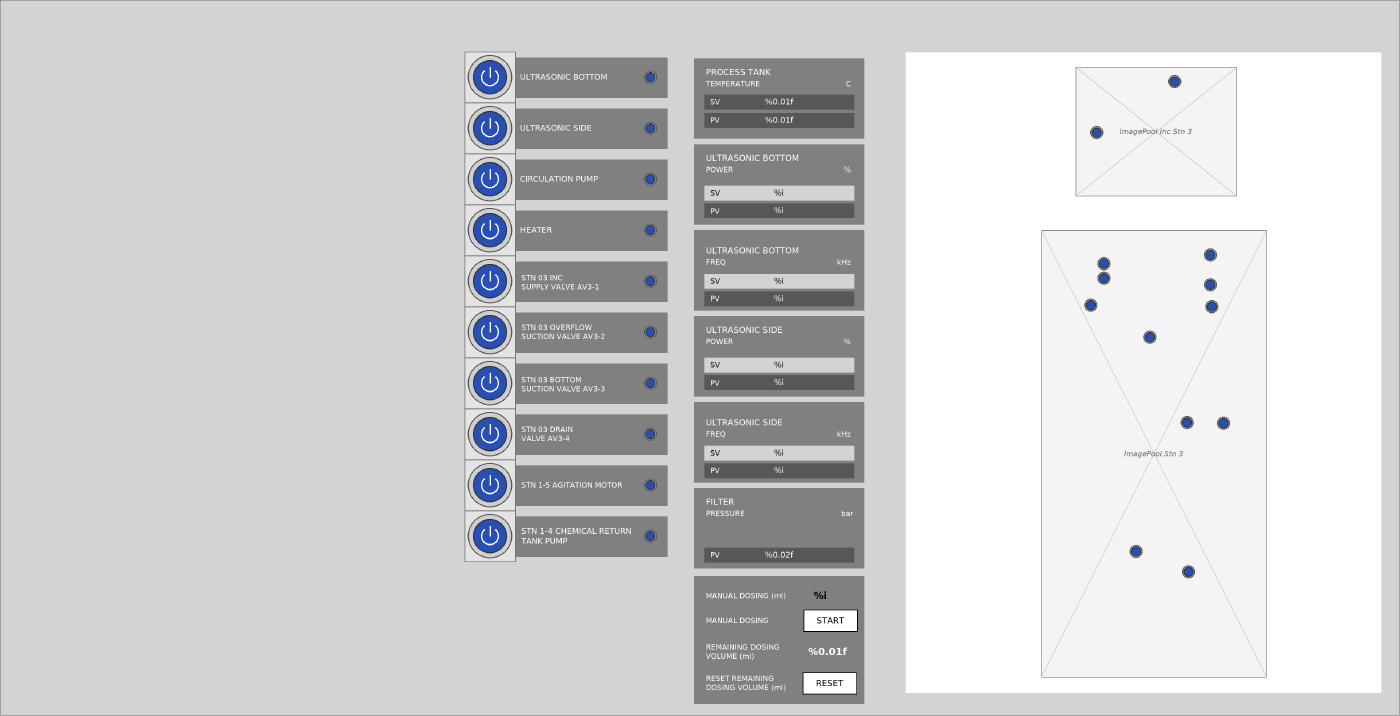
VISUALIZATION Manual_Station03  // 1920x983
    Rectangle (0,0 1920x983)
    Rectangle (1242,72 652x879)
    Image (1428,316 309x614), image: ImagePool.Stn 3
    RoundedRectangle (676,79 239x55)
    Label (710,98 163x16), "ULTRASONIC BOTTOM"
    Lamp1 (882,96 20x20), variable: ARdsMAP_HmiVariableStn[3].bProTankUsBtm_IND, style: Lamp-Lamp1-Blue
    PowerSwitch (637,71 70x70), variable: ARdsMAP_HmiVariableStn[3].bProTankUsBtm_PB, behaviour: TOGGLE, style: Switch-PowerSwitch-Blue
    RoundedRectangle (684,219 231x55)
    Label (710,238 151x16), "CIRCULATION PUMP"
    Lamp1 (882,236 20x20), variable: ARdsMAP_HmiVariableStn[3].bProTankPump_IND, style: Lamp-Lamp1-Blue
    PowerSwitch (637,211 70x70), variable: ARdsMAP_HmiVariableStn[3].bProTankPump_PB, behaviour: TOGGLE, style: Switch-PowerSwitch-Blue
    RoundedRectangle (684,289 231x55)
    Label (710,308 151x16), "HEATER"
    Lamp1 (882,306 20x20), variable: ARdsMAP_HmiVariableStn[3].bProTankHeater_IND, style: Lamp-Lamp1-Blue
    PowerSwitch (637,281 70x70), variable: ARdsMAP_HmiVariableStn[3].bProTankHeater_PB, behaviour: TOGGLE, style: Switch-PowerSwitch-Blue
    RoundedRectangle (676,149 239x55)
    Label (710,168 163x16), "ULTRASONIC SIDE"
    Lamp1 (882,166 20x20), variable: ARdsMAP_HmiVariableStn[3].bProTankUsSide_IND, style: Lamp-Lamp1-Blue
    PowerSwitch (637,141 70x70), variable: ARdsMAP_HmiVariableStn[3].bProTankUsSide_PB, behaviour: TOGGLE, style: Switch-PowerSwitch-Blue
    RoundedRectangle (684,429 231x55)
    Label (712,438 160x36), "STN 03 OVERFLOW SUCTION VALVE AV3-2"
    Lamp1 (882,446 20x20), variable: ARdsMAP_HmiVariableStn[3].bValve02_IND, style: Lamp-Lamp1-Blue
    PowerSwitch (637,421 70x70), variable: ARdsMAP_HmiVariableStn[3].bValve02_PB, behaviour: TOGGLE, style: Switch-PowerSwitch-Blue
    RoundedRectangle (684,359 231x55)
    Lamp1 (882,376 20x20), variable: ARdsMAP_HmiVariableStn[3].bValve01_IND, style: Lamp-Lamp1-Blue
    PowerSwitch (637,351 70x70), variable: ARdsMAP_HmiVariableStn[3].bValve01_PB, behaviour: TOGGLE, style: Switch-PowerSwitch-Blue
    Label (712,370 151x36), "STN 03 INC SUPPLY VALVE AV3-1"
    RoundedRectangle (684,569 231x55)
    Label (712,578 160x36), "STN 03 DRAIN VALVE AV3-4"
    Lamp1 (882,586 20x20), variable: ARdsMAP_HmiVariableStn[3].bValve04_IND, style: Lamp-Lamp1-Blue
    PowerSwitch (637,561 70x70), variable: ARdsMAP_HmiVariableStn[3].bValve04_PB, behaviour: TOGGLE, style: Switch-PowerSwitch-Blue
    RoundedRectangle (684,499 231x55)
    Lamp1 (882,516 20x20), variable: ARdsMAP_HmiVariableStn[3].bValve03_IND, style: Lamp-Lamp1-Blue
    PowerSwitch (637,491 70x70), variable: ARdsMAP_HmiVariableStn[3].bValve03_PB, behaviour: TOGGLE, style: Switch-PowerSwitch-Blue
    Label (712,510 151x36), "STN 03 BOTTOM SUCTION VALVE AV3-3"
    RoundedRectangle (684,639 231x55)
    Label (712,648 160x36), "STN 1-5 AGITATION MOTOR"
    Lamp1 (882,656 20x20), variable: ARdsMAP_HmiVariableGeneral.bProTankAgitationMotor_IND, style: Lamp-Lamp1-Blue
    PowerSwitch (637,631 70x70), variable: ARdsMAP_HmiVariableGeneral.bProTankAgitationMotor_PB, behaviour: TOGGLE, style: Switch-PowerSwitch-Blue
    RoundedRectangle (684,709 231x55)
    Label (712,718 160x36), "STN 1-4 CHEMICAL RETURN TANK PUMP"
    Lamp1 (882,726 20x20), variable: ARdsMAP_HmiVariableGeneral.bProTankPump_IND, style: Lamp-Lamp1-Blue
    PowerSwitch (637,701 70x70), variable: ARdsMAP_HmiVariableGeneral.bProTankPump_PB, behaviour: TOGGLE, style: Switch-PowerSwitch-Blue
    Lamp1 (1567,453 20x20), variable: ARdsMAP_HmiVariableStn[3].bProTankUsBtm_IND, style: Lamp-Lamp1-Blue
    Lamp1 (1548,747 20x20), variable: ARdsMAP_HmiVariableStn[3].bProTankPump_IND, style: Lamp-Lamp1-Blue
    Lamp1 (1504,372 20x20), variable: ARdsMAP_HmiVariableStn[3].bProTankHeater_IND, style: Lamp-Lamp1-Blue
    Lamp1 (1486,409 20x20), variable: ARdsMAP_HmiVariableStn[3].bProTankUsSide_IND, style: Lamp-Lamp1-Blue
    Lamp1 (1668,571 20x20), variable: ARdsMAP_HmiVariableStn[3].bValve02_IND, style: Lamp-Lamp1-Blue
    Lamp1 (1620,775 20x20), variable: ARdsMAP_HmiVariableStn[3].bValve04_IND, style: Lamp-Lamp1-Blue
    Lamp1 (1618,570 20x20), variable: ARdsMAP_HmiVariableStn[3].bValve03_IND, style: Lamp-Lamp1-Blue
    Lamp1 (1650,340 20x20), variable: ARdsMAP_HmiVariableStn[3].bOverflowMaxLevel_IND, style: Lamp-Lamp1-Blue
    Lamp1 (1504,352 20x20), variable: ARdsMAP_HmiVariableStn[3].bProcessTankMinLevel_IND, style: Lamp-Lamp1-Blue
    Lamp1 (1650,381 20x20), variable: ARdsMAP_HmiVariableStn[3].bOverflowMinLevel_IND, style: Lamp-Lamp1-Blue
    Lamp1 (1652,411 20x20), variable: ARdsMAP_HmiVariableStn[3].bProTankUsSide_IND, style: Lamp-Lamp1-Blue
    Image (1475,92 221x177), image: ImagePool.Inc Stn 3
    Lamp1 (1601,102 20x20), variable: ARdsMAP_HmiVariableStn[3].bValve01_IND, style: Lamp-Lamp1-Blue
    Lamp1 (1494,172 20x20), variable: ARdsMAP_HmiVariableStn[3].bDosingPump_IND, style: Lamp-Lamp1-Blue
    Group (952,791 233x175)
        RoundedRectangle (0,0 233x175)
        Rectangle (150,46 74x30), "START", colour toggle: ARbStnManualDosingST[3]
            toggle ARbStnManualDosingST[3]
        Label (13,47 109x28), "MANUAL DOSING"
        Label (13,13 121x28), "MANUAL DOSING (ml)"
        Rectangle (132,13 82x28), "%i", text variable: ARDSProminentDosingHMI[3].In_iManualDosingVolume_ml
            OnMouseDown: write the text variable via VisuDialogs.Numpad, min 1, max 32767
        Label (13,133 129x28), "RESET REMAINING DOSING VOLUME (ml)"
        Rectangle (149,132 74x30), "RESET", colour toggle: ARDSProminentDosingHMI[3].In_bResetRemainedDosingVolumePB
            tap ARDSProminentDosingHMI[3].In_bResetRemainedDosingVolumePB
        Label (13,90 118x28), "REMAINING DOSING VOLUME (ml)"
        Rectangle (142,90 82x28), "%0.01f", text variable: ARDSProminentDosingHMI[3].Out_rRemainedDosingVolume_ml
    Group (952,80 233x110)
        RoundedRectangle (0,0 233x110)
        Label (189,24 29x22), "C"
        Rectangle (14,50 205x20), "%0.01f", text variable: ARrStnTempSV[3]
        Label (19,49 22x22), "SV"
        Rectangle (14,75 205x20), "%0.01f", text variable: ARrStnTempPV[3]
        Label (19,74 22x22), "PV"
        Label (13,11 150x16), "PROCESS TANK"
        Label (13,24 99x22), "TEMPERATURE"
    Group (952,198 233x110)
        RoundedRectangle (0,0 233x110)
        Label (189,24 29x22), "%"
        Rectangle (14,57 205x20), "%i", text variable: ARiStnManualUSBtmAsv[3]
            OnMouseDown: write the text variable via VisuDialogs.Numpad, min 10, max 100
        Label (19,56 22x22), "SV"
        Rectangle (14,81 205x20), "%i", text variable: ARiStnUSBtmAPv[3]
        Label (19,81 22x22), "PV"
        Label (13,11 150x16), "ULTRASONIC BOTTOM"
        Label (13,24 99x22), "POWER"
    Group (952,670 233x110)
        RoundedRectangle (0,0 233x110)
        Label (189,24 32x22), "bar"
        Rectangle (14,82 205x20), "%0.02f", text variable: ARrStnFilterPressurePV[3]
        Label (19,81 22x22), "PV"
        Label (13,11 150x16), "FILTER"
        Label (13,24 99x22), "PRESSURE"
    Group (952,316 233x110)
        RoundedRectangle (0,0 233x110)
        Label (189,33 29x22), "kHz"
        Rectangle (14,84 205x20), "%i", text variable: ARiStnUSBtmAFreqPv[3]
        Label (19,83 22x22), "PV"
        Rectangle (14,60 205x20), "%i", text variable: DSWeberEnclosure[1].DSWeberGenerator[6].DSWeberMulFreqSwitching.iFreqOutput_TS
            tap DSWeberEnclosure[1].DSWeberGenerator[6].DSWeberMulFreqSwitching.bFreqSwitchingPB_TS
        Label (19,59 22x22), "SV"
        Label (13,33 99x22), "FREQ"
        Label (13,20 150x16), "ULTRASONIC BOTTOM"
    Group (952,434 233x110)
        RoundedRectangle (0,0 233x110)
        Label (189,24 29x22), "%"
        Rectangle (14,57 205x20), "%i", text variable: ARiStnManualUSSideAsv[3]
            OnMouseDown: write the text variable via VisuDialogs.Numpad, min 10, max 100
        Label (19,56 22x22), "SV"
        Rectangle (14,81 205x20), "%i", text variable: ARiStnUSSideAPv[3]
        Label (19,81 22x22), "PV"
        Label (13,11 150x16), "ULTRASONIC SIDE"
        Label (13,24 99x22), "POWER"
    RoundedRectangle (952,552 233x110)
    Label (965,585 99x22), "FREQ"
    Label (965,572 150x16), "ULTRASONIC SIDE"
    Label (1141,585 29x22), "kHz"
    Rectangle (966,636 205x20), "%i", text variable: ARiStnUSSideAFreqPv[3]
    Label (971,635 22x22), "PV"
    Rectangle (966,612 205x20), "%i", text variable: DSWeberEnclosure[1].DSWeberGenerator[5].DSWeberMulFreqSwitching.iFreqOutput_TS
        tap DSWeberEnclosure[1].DSWeberGenerator[5].DSWeberMulFreqSwitching.bFreqSwitchingPB_TS
    Label (971,611 22x22), "SV"
END_VISUALIZATION

(* stored: Version 1.1.0.1, ProductVersion 3.1.4024.12
   Visu Manual_Station03: Id {4ad16970-347f-4154-ad07-1e9b9a19f299} *)
